{attribute 'qualified_only'}
{attribute 'strict'}
{attribute 'to_string'}
TYPE E_ServiceCallSubmitResult :
(
	Queued := 0,
	CallerNotConfigured := 1,
	CoordinatorNotReady := 2,
	UnknownService := 3,
	DependencyNotDeclared := 4,
	NotOwner := 5,
	Busy := 6,
	InvalidCommand := 7,
	ParameterSizeMismatch := 8,
	ParameterTypeResolutionFailed := 9,
	ParameterTypeMismatch := 10
) UDINT;
END_TYPE

(* stored: Version 1.1.0.1, ProductVersion 3.1.4026.18
   DUT E_ServiceCallSubmitResult: Id {cdc3d458-02c9-457a-9417-1768c12cdc06} *)
